ABB RobotStudio station: Lab1.4_20210903-152520.rsstn

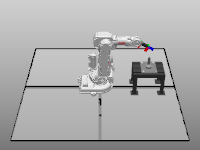
Station Lab1.2 (saved by RobotStudio 21.2.9526.0)
Controller IRB140
  mechanical unit ROB_1: IRB140_6_81_C_03_3, 6 joints, base frame (0, 0, 0) mm
Layout (positions relative to the parent item):
  - IRB140_6_81_C_03_3 [mechanism, from Robots\IRB140_6_81_C_G_03.rslib] at (0, 0, 0) mm; joint values [0, 0, 0, 0, 0.5236, 0] (rad or m)
  - UISpenholder [mechanism, from RS1\UISpenholder.rslib] at (506.29, 0, 679.5) mm, rotated rx 180 ry 60 rz 180 deg
  - table_and_fixture_140 [part, from Training Objects\propeller_table.rslib] at (400, -175, 0) mm
Attachment: UISpenholder is attached to IRB140_6_81_C_03_3 / Link6
Targets, tools, work objects and paths stored in the station, written as RAPID:
! task T_ROB1
MODULE CalibData
  PERS tooldata UISpenholder:=[TRUE,[[0,0,110],[1,0,0,0]],[1,[0,0,1],[1,0,0,0],0,0,0]];
ENDMODULE

